{attribute 'linkalways'} 
{attribute 'no_explicit_call' := 'This FB is a CLASS and must be accessed using methods or properties'}
{attribute 'enable_dynamic_creation'}
FUNCTION_BLOCK FINAL MIN_BYTE EXTENDS Node
VAR
	in1 : _BYTE(0);
	in2 : _BYTE(0);
	out : _BYTE(0);
END_VAR

METHOD PUBLIC Clone : I_Node
VAR
	pNode : POINTER TO MIN_BYTE;
END_VAR
pNode := __NEW(MIN_BYTE);
Clone := pNode^;
END_METHOD

METHOD FB_init : BOOL
VAR_INPUT
	bInitRetains : BOOL; // if TRUE, the retain variables are initialized (warm start / cold start)
	bInCopyCode : BOOL;  // if TRUE, the instance afterwards gets moved into the copy code (online change)
END_VAR
AddInput('in1',THIS^.in1);
AddInput('in2',THIS^.in2);
AddOutput('out', THIS^.out);
END_METHOD

METHOD PROTECTED OnExecute
VAR
END_VAR
out.Value := MIN(in1.Value, in2.Value);
END_METHOD

END_FUNCTION_BLOCK

(* stored: Version 1.1.0.1, ProductVersion 3.1.4024.15
   POU MIN_BYTE: Id {f2d4426c-89d0-42cc-8284-0ecaf2f22651}, SpecialFunc None
   Folder Constructor: Id {aafbef08-e8c5-4eb4-adbd-20f3805f4cba}
   Method Clone: Id {0aaba451-cae3-4e1b-b9f1-f28bf7abcf28}
   Method FB_init: Id {0051d3c9-94fa-4e97-a24e-5976f6b43fd7}
   Method OnExecute: Id {332e2840-07d6-43ca-bb6f-567827fee311} *)
